// TIA Portal V19 export
DATA_BLOCK "GETIO_PAC3220"   // DB12
// stored: InstanceOfName GETIO, OfSystemLibElement GETIO, OfSystemLibVersion 1.1
"GETIO"
   // VAR_INPUT
   //    ID : HW_SUBMODULE;
   // END_VAR
   // VAR_OUTPUT
   //    STATUS : DWord;
   //    LEN : Int;
   // END_VAR
   // VAR_IN_OUT
   //    INPUTS : Variant;
   // END_VAR
BEGIN
END_DATA_BLOCK
